// TIA Portal V16 export
// export: Created 2021-07-12T14:47:17.9161173Z, ExportSetting WithDefaults, DisplayName Totally Integrated Automation Portal, DisplayVersion V16, DisplayName TIA Portal Version Control Interface, DisplayVersion V16, DisplayName TIA Portal Openness, DisplayVersion V16, DisplayName STEP 7 Professional, DisplayVersion V16, DisplayName STEP 7 Safety, DisplayVersion V16, DisplayName WinCC Professional, DisplayVersion V16
TYPE "LSimaHydTO_typeInternalControlForceCmd"
TITLE = LSimaHydTO_typeInternalControlForceCmd
// Defines force command
// stored: IsFailsafeCompliant false
   STRUCT
      mode : DInt;   // 0: deactivate / 1: activate immediately / 2: starting from the time a condition is met.
      forceProfileMode : DInt;   // 0: with force value / 1: profile is a function of time / 2: profile is a function of position
      conditionMode : DInt := 1;   // 1: based on time / 2: based on position / 3: based on force/pressure
      compareMode : DInt := 1;   // 1: Value greater than or equal to ConditionValue / 2: Value less than ConditionValue
      conditionValue : LReal;   // comparison value for switching condition
      clampingMonitoring : Bool;   // TRUE: end stop detection is activated, motion stops after detection
      followingErrorDeviation : LReal;   // Required following error for recognition of the endstop
      forceValue : LReal;   // Force setpoint
      forceRamp : LReal;   // Force setpoint increase
      velocityLimitingValue : LReal;   // Rate limiting value during pressure control, the dynamic response of the pressure Value > 0.0 Use the specified value
      commandID : UDInt;   // commanID for tracking
   END_STRUCT;
END_TYPE
